(* Logix 5000 project; controller RN21_Architecture 1769-L16ER-BB1B rev 35.11; software revision 35.00 *)
// For Developing the Arch

TASK MainTask (continuous, watchdog 500 ms) : MainProgram

MODULES
   Local : 1769-L16ER-BB1B (PointIO 0, rev 35.11)
      Discrete_IO : Embedded (PointIO 1, rev 35.11, Output RPI 20 ms)
END_MODULES

TYPE UDT_Alarm :
STRUCT
   ALM_YearValue : INT;
   ALM_MonthValue : INT;
   ALM_DayValue : INT;
   ALM_HourValue : INT;
   ALM_MinuteValue : INT;
   ALM_SecondValue : INT;
   ALM_ActionId : INT;
   ALM_Reason : INT;
   ALM_AlarmId1 : DINT;
   ALM_AlarmId2 : DINT;
   ALM_AlarmId3 : DINT;
   ALM_AlarmId4 : DINT;
   ALM_AlarmId5 : DINT;
   ALM_AlarmId6 : DINT;
   ALM_AlarmId7 : DINT;
END_STRUCT
END_TYPE

TYPE UDT_Audit :
STRUCT
   AUD_YearValue : INT;
   AUD_MonthValue : INT;
   AUD_DayValue : INT;
   AUD_HourValue : INT;
   AUD_MinuteValue : INT;
   AUD_SecondValue : INT;
   AUD_ActionId : INT;
   AUD_ReasonId : INT;
   AUD_OldValue : REAL;
   AUD_NewValue : REAL;
   AUD_AppUserId : STRING;
END_STRUCT
END_TYPE

TYPE UDT_Batch :
STRUCT
   BMAN_YearValue : INT;
   BMAN_MonthValue : INT;
   BMAN_DayValue : INT;
   BMAN_HourValue : INT;
   BMAN_MinuteValue : INT;
   BMAN_SecondValue : INT;
   BMAN_BATCH_SIZE : REAL;
   BMAN_BatchStatus : INT;
   BMAN_EXPIR_DATE : INT;
   BMAN_MANFACT_DATE : INT;
   BMAN_EXPIRY_MONTH : INT;
   BMAN_EXPIRY_YEAR : INT;
   BMAN_MANFACT_MONTH : INT;
   BMAN_MANFACT_YEAR : INT;
   BMAN_BATCH_RECIPENAME : STRING;
   BMAN_OPERATOR_CODE : STRING;
   BMAN_PROGRAM_NO : STRING;
   BMAN_TAG_NO : STRING;
   BMAN_LOT_NO : STRING;
   BMAN_PRODUCT_CODE : STRING;
   BMAN_PRODUCT_NAME : STRING;
   BMAN_BATCH_NO : STRING;
END_STRUCT
END_TYPE

TYPE UDT_Login :
STRUCT
   LOGIN_YearValue : INT;
   LOGIN_MonthValue : INT;
   LOGIN_DayValue : INT;
   LOGIN_HourValue : INT;
   LOGIN_MinuteValue : INT;
   LOGIN_SecondValue : INT;
   LOGIN_Reason : INT;
   LOGIN_LoginReason : INT;
   LOGIN_AppUserId : STRING;
END_STRUCT
END_TYPE

TYPE UDT_Process :
STRUCT
   PDL_Year : INT;
   PDL_Month : INT;
   PDL_Date : INT;
   PDL_Hour : INT;
   PDL_Minute : INT;
   PDL_Second : INT;
   PDL_Reason : INT;
   PDL_ActionId : INT;
   PDL_ProcessStatus : INT;
   PDL_CYCLEID : INT;
   PDL_ProcessData : REAL[20];
END_STRUCT
END_TYPE

TYPE UDT_Recipe :
STRUCT
   RP_Year : INT;
   RP_Month : INT;
   RP_Date : INT;
   RP_Hour : INT;
   RP_Minute : INT;
   RP_Second : INT;
   RP_PRINT_INTERVAL : INT;
   RP_CYCLE_ID : INT;
   RP_RecipeData1 : REAL[50];
   RP_RecipeData2 : DINT[50];
END_STRUCT
END_TYPE

ADD_ON_INSTRUCTION AOI_ALM_Arch   (* revision 1.0 *)
VAR_INPUT
   FBI_DataLogTrig : BOOL; {required}   // Trigger Bit for Data Log Generation
END_VAR
VAR_IN_OUT
   FBO_TriggerBit : BOOL; {required}   // Server Trigger Bit
   FBIO_Src : UDT_Alarm; {required}   // Source UDT Data
   FBIO_Ser : UDT_Alarm; {required}   // Server UDT Data
END_VAR
VAR_INPUT
   FBI_PLCServerCommFailed : BOOL; {access None, required}   // PLC to Server Communication Fail Timer Done
END_VAR
VAR_IN_OUT
   FBIO_SerUniqueNum : DINT; {required}   // Server Unique Number(Server UID)
   FBIO_SrcUniqueNum : DINT; {required}   // Source Unique Number (PLC UID)
END_VAR
VAR
   FBL_Prim : UDT_Alarm; {access None}   // Primary UDT Data
   FBL_Buff : UDT_Alarm[100]; {access None}   // Buffer UDT Data
   FBL_Sec : UDT_Alarm; {access None}   // Secondary UDT Data
   FBL_IndexStore : DINT; {access None}   // Index Store Value
   FBL_Bit4 : BOOL; {access None}   // Source to Primary Moved
   FBL_TMR2 : TIMER := (PRE := 1, ACC := 1); {access None}   // Source UID Reset Delay
   FBL_Bit1 : BOOL; {access None}   // Source UID Reseted
   FBL_Bit2 : BOOL; {access None}   // Source UID Less than Server UID
   FBL_Bit6 : BOOL; {access None}   // Data Moving From Secondary to Server
   FBL_TMR3 : TIMER := (PRE := 5000, ACC := 5); {access None}   // Load Movement Delay
   FBL_Bit5 : BOOL; {access None}   // Data Load From Buffer to Secondary Flag
   FBL_IndexLoad : DINT; {access None}   // Index Load Value
   FBL_Bit3 : BOOL; {access None}   // Buffer to Secondary Moved
   FBL_TMR1 : TIMER := (PRE := 5000); {access None}   // Server UID Movement Delay
   FBL_PrimUniqueNum : DINT; {access None}   // Primary Unique Number (PLC UID)
   FBL_BuffUniqueNum : DINT[100]; {access None}   // Buffer Unique Number (PLC UID)
   FBL_SecUniqueNum : DINT; {access None}   // Secondary Unique Number (PLC UID)
   FBL_ONS : DINT; {access None}   // Common ONS DINT
END_VAR

ROUTINE Logic   (* ladder *)
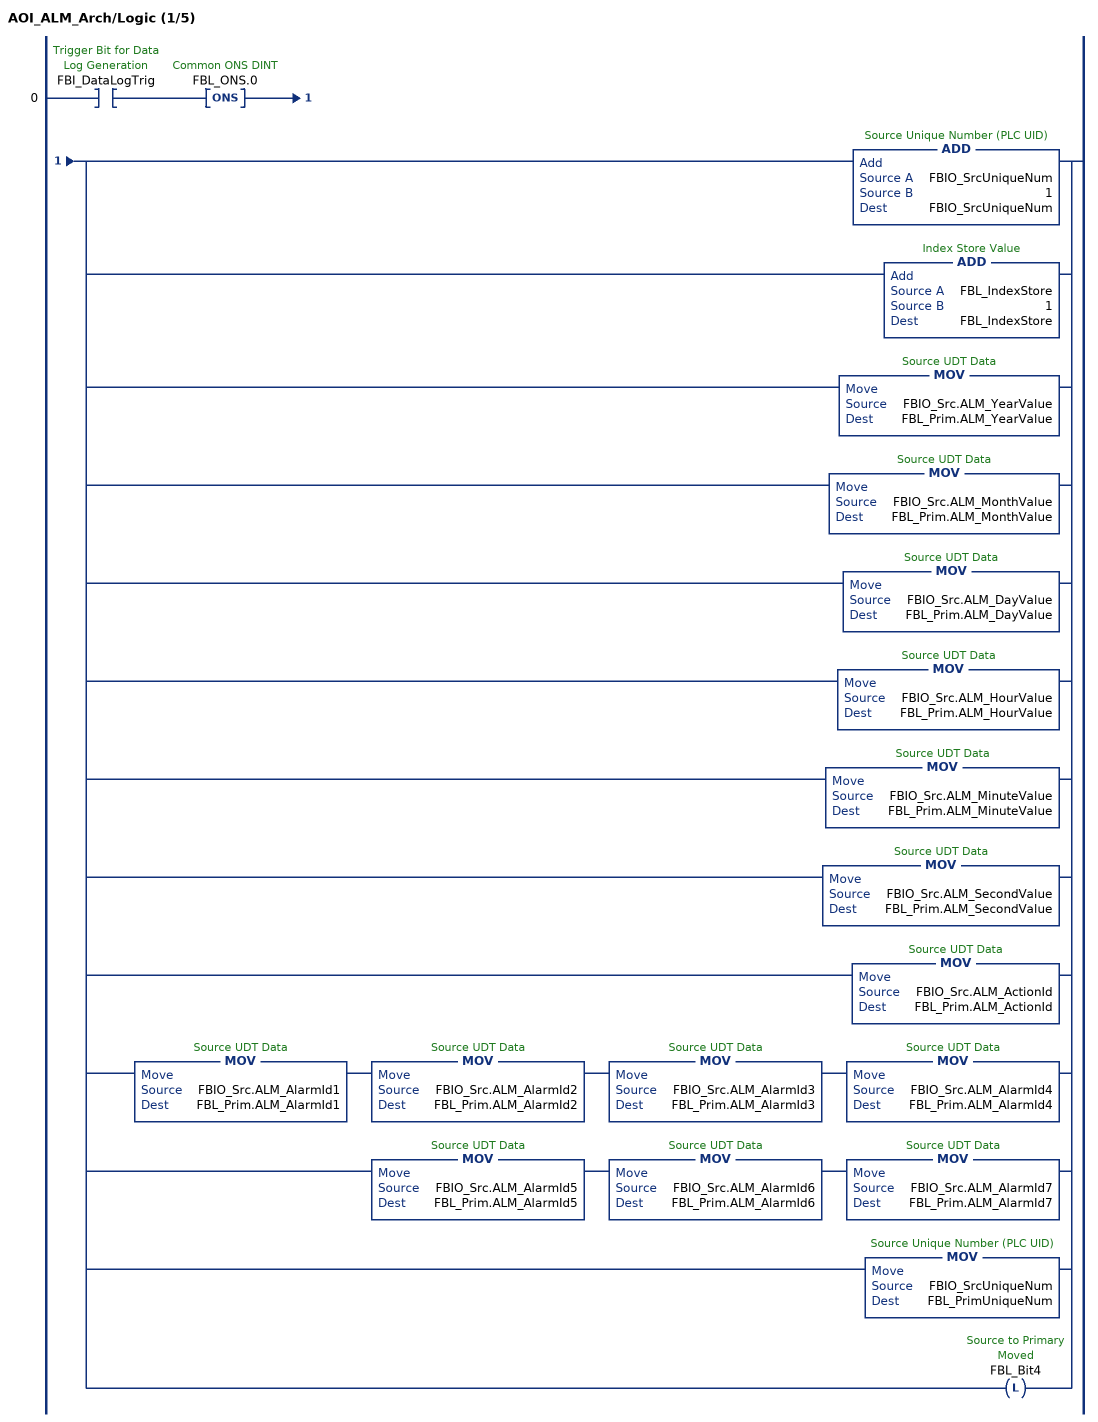
   0: XIC(FBI_DataLogTrig)ONS(FBL_ONS.0)[ADD(FBIO_SrcUniqueNum,1,FBIO_SrcUniqueNum) ,ADD(FBL_IndexStore,1,FBL_IndexStore) ,MOV(FBIO_Src.ALM_YearValue,FBL_Prim.ALM_YearValue) ,MOV(FBIO_Src.ALM_MonthValue,FBL_Prim.ALM_MonthValue) ,MOV(FBIO_Src.ALM_DayValue,FBL_Prim.ALM_DayValue) ,MOV(FBIO_Src.ALM_HourValue,FBL_Prim.ALM_HourValue) ,MOV(FBIO_Src.ALM_MinuteValue,FBL_Prim.ALM_MinuteValue) ,MOV(FBIO_Src.ALM_SecondValue,FBL_Prim.ALM_SecondValue) ,MOV(FBIO_Src.ALM_ActionId,FBL_Prim.ALM_ActionId) ,MOV(FBIO_Src.ALM_AlarmId1,FBL_Prim.ALM_AlarmId1) MOV(FBIO_Src.ALM_AlarmId2,FBL_Prim.ALM_AlarmId2) MOV(FBIO_Src.ALM_AlarmId3,FBL_Prim.ALM_AlarmId3) MOV(FBIO_Src.ALM_AlarmId4,FBL_Prim.ALM_AlarmId4) ,MOV(FBIO_Src.ALM_AlarmId5,FBL_Prim.ALM_AlarmId5) MOV(FBIO_Src.ALM_AlarmId6,FBL_Prim.ALM_AlarmId6) MOV(FBIO_Src.ALM_AlarmId7,FBL_Prim.ALM_AlarmId7) ,MOV(FBIO_SrcUniqueNum,FBL_PrimUniqueNum) ,OTL(FBL_Bit4) ];
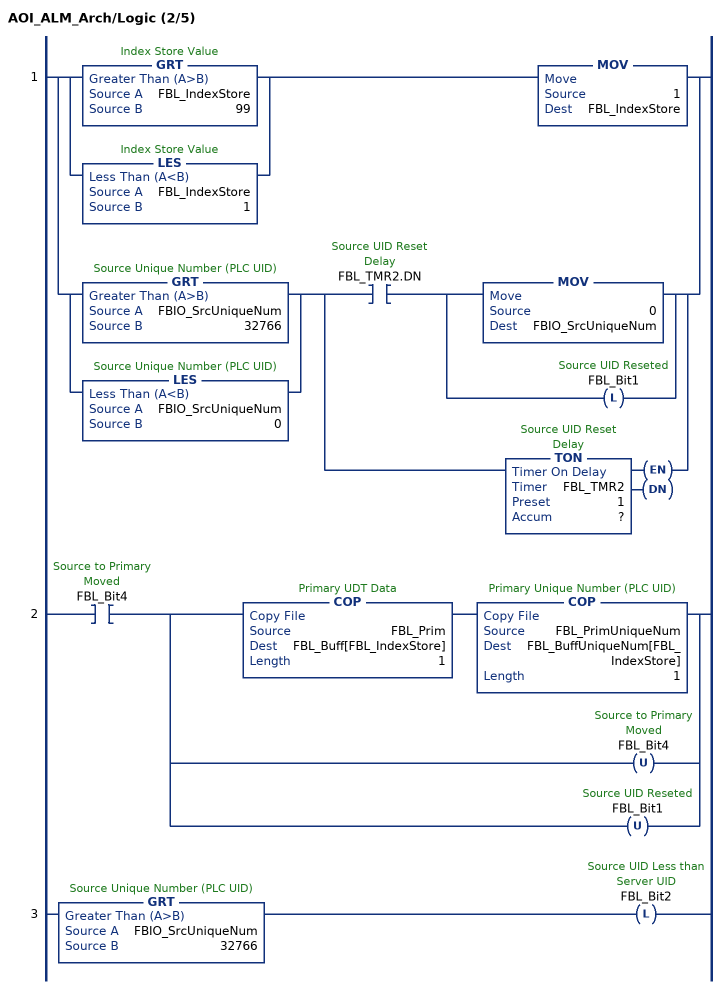
   1: [[GRT(FBL_IndexStore,99) ,LES(FBL_IndexStore,1) ] MOV(1,FBL_IndexStore) ,[GRT(FBIO_SrcUniqueNum,32766) ,LES(FBIO_SrcUniqueNum,0) ] [XIC(FBL_TMR2.DN) [MOV(0,FBIO_SrcUniqueNum) ,OTL(FBL_Bit1) ] ,TON(FBL_TMR2,?,?) ] ];
   2: XIC(FBL_Bit4)[COP(FBL_Prim,FBL_Buff[FBL_IndexStore],1) COP(FBL_PrimUniqueNum,FBL_BuffUniqueNum[FBL_IndexStore],1) ,OTU(FBL_Bit4) ,OTU(FBL_Bit1) ];
   3: GRT(FBIO_SrcUniqueNum,32766)OTL(FBL_Bit2);
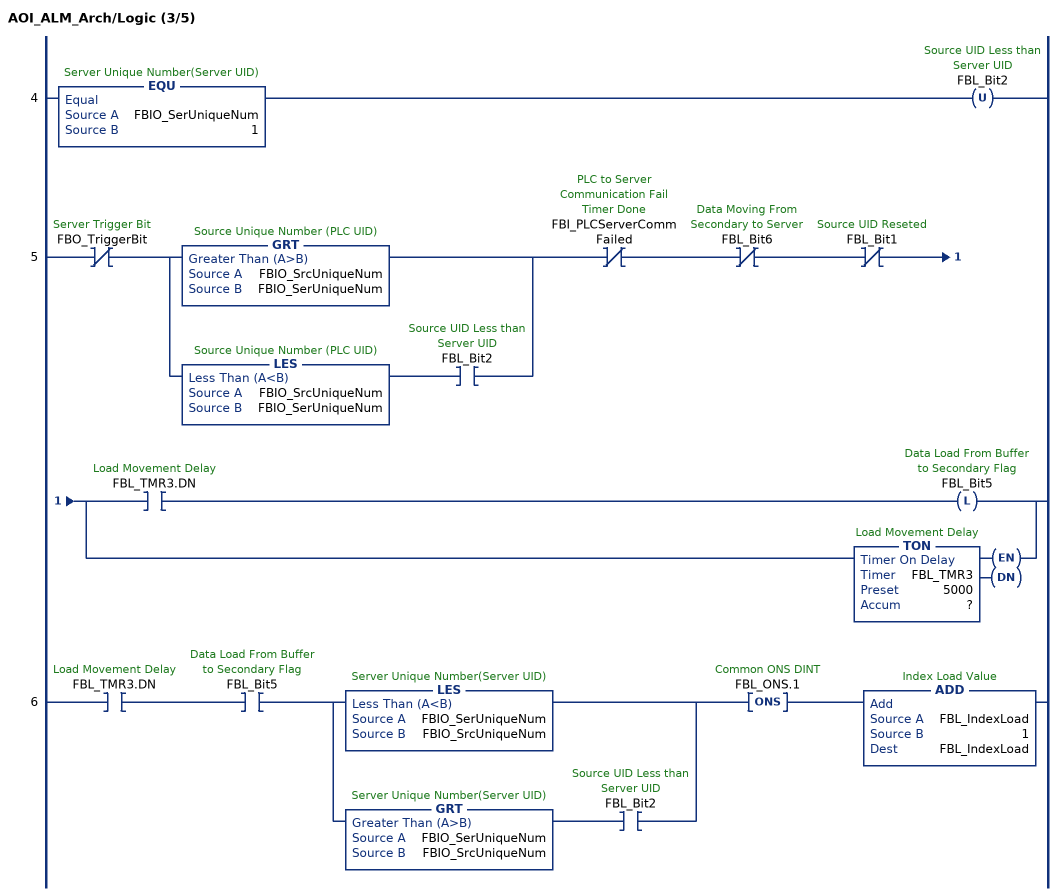
   4: EQU(FBIO_SerUniqueNum,1)OTU(FBL_Bit2);
   5: XIO(FBO_TriggerBit)[GRT(FBIO_SrcUniqueNum,FBIO_SerUniqueNum) ,LES(FBIO_SrcUniqueNum,FBIO_SerUniqueNum) XIC(FBL_Bit2) ]XIO(FBI_PLCServerCommFailed)XIO(FBL_Bit6)XIO(FBL_Bit1)[XIC(FBL_TMR3.DN) OTL(FBL_Bit5) ,TON(FBL_TMR3,?,?) ];
   6: XIC(FBL_TMR3.DN)XIC(FBL_Bit5)[LES(FBIO_SerUniqueNum,FBIO_SrcUniqueNum) ,GRT(FBIO_SerUniqueNum,FBIO_SrcUniqueNum) XIC(FBL_Bit2) ]ONS(FBL_ONS.1)ADD(FBL_IndexLoad,1,FBL_IndexLoad);
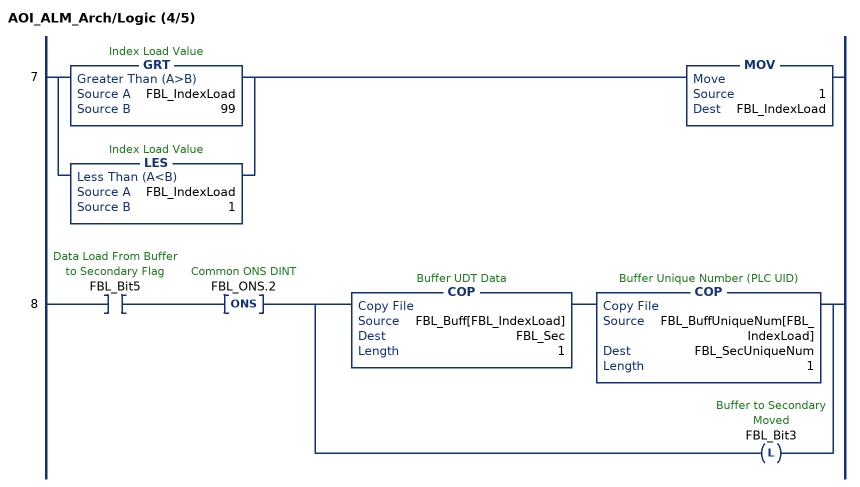
   7: [GRT(FBL_IndexLoad,99) ,LES(FBL_IndexLoad,1) ]MOV(1,FBL_IndexLoad);
   8: XIC(FBL_Bit5)ONS(FBL_ONS.2)[COP(FBL_Buff[FBL_IndexLoad],FBL_Sec,1) COP(FBL_BuffUniqueNum[FBL_IndexLoad],FBL_SecUniqueNum,1) ,OTL(FBL_Bit3) ];
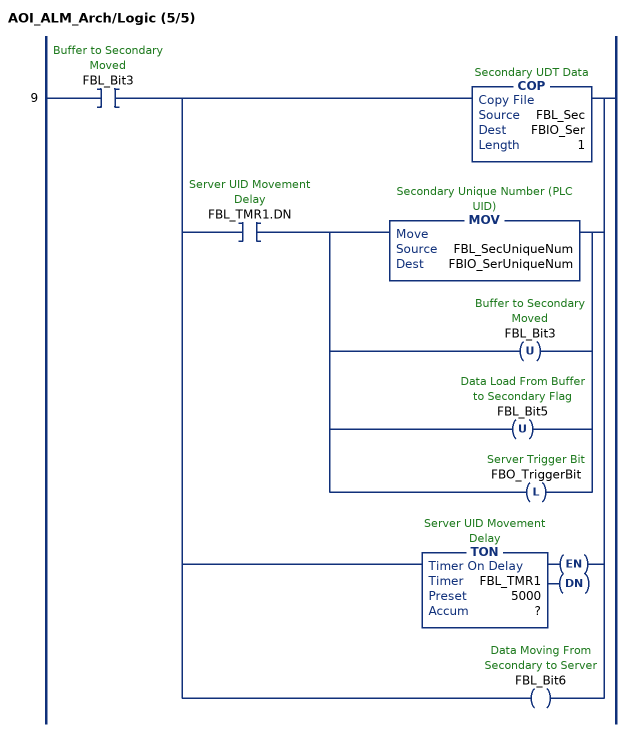
   9: XIC(FBL_Bit3)[COP(FBL_Sec,FBIO_Ser,1) ,XIC(FBL_TMR1.DN) [MOV(FBL_SecUniqueNum,FBIO_SerUniqueNum) ,OTU(FBL_Bit3) ,OTU(FBL_Bit5) ,OTL(FBO_TriggerBit) ] ,TON(FBL_TMR1,?,?) ,OTE(FBL_Bit6) ];
END_ROUTINE
END_ADD_ON_INSTRUCTION

ADD_ON_INSTRUCTION AOI_ALM_DataCapture   (* revision 1.0 *)
// Alarm Data Capture logic
VAR_INPUT
   FBI_AlarmTag : BOOL; {required}
END_VAR
VAR_OUTPUT
   FBO_AlarmPosID : BOOL; {access Read Only, required}
   FBO_ALM_Trig : BOOL; {required}
END_VAR
VAR
   FBL_PosTrig : BOOL; {access None}
   FBL_NegTrig : BOOL; {access None}
   ONS : DINT; {access None}
END_VAR

ROUTINE Logic   (* ladder *)
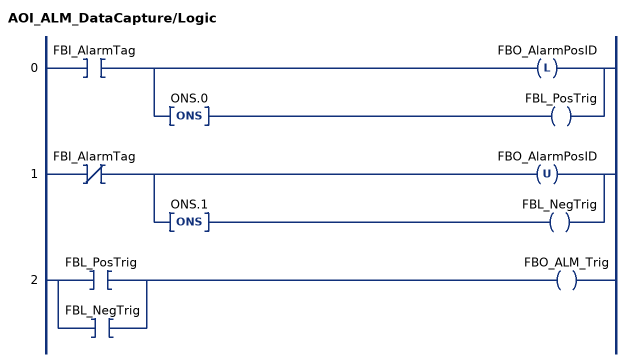
   0: XIC(FBI_AlarmTag)[OTL(FBO_AlarmPosID) ,ONS(ONS.0) OTE(FBL_PosTrig) ];
   1: XIO(FBI_AlarmTag)[OTU(FBO_AlarmPosID) ,ONS(ONS.1) OTE(FBL_NegTrig) ];
   2: [XIC(FBL_PosTrig) ,XIC(FBL_NegTrig) ]OTE(FBO_ALM_Trig);
END_ROUTINE
END_ADD_ON_INSTRUCTION

ADD_ON_INSTRUCTION AOI_AUD_Arch   (* revision 1.0 *)
VAR_INPUT
   FBI_DataLogTrig : BOOL; {required}   // Trigger Bit for Data Log Generation
END_VAR
VAR_IN_OUT
   FBO_TriggerBit : BOOL; {required}   // Server Trigger Bit
   FBIO_Src : UDT_Audit; {required}   // Source UDT Data
   FBIO_Ser : UDT_Audit; {required}   // Server UDT Data
END_VAR
VAR_INPUT
   FBI_PLCServerCommFailed : BOOL; {access None, required}   // PLC to Server Communication Fail Timer Done
END_VAR
VAR_IN_OUT
   FBIO_SrcUniqueNum : DINT; {required}   // Source Unique Number(PLC UID)
   FBIO_SerUniqueNum : DINT; {required}   // Server Unique Number(PLC UID)
END_VAR
VAR
   FBL_Prim : UDT_Audit; {access None}   // Primary UDT Data
   FBL_Buff : UDT_Audit[100]; {access None}   // Buffer UDT Data
   FBL_Sec : UDT_Audit; {access None}   // Secondary UDT Data
   FBL_IndexStore : DINT; {access None}   // Index Store Value
   FBL_Bit4 : BOOL; {access None}   // Primary Movement Completed
   FBL_TMR2 : TIMER := (PRE := 1, ACC := 1); {access None}   // Source UID Reset Delay
   FBL_Bit1 : BOOL; {access None}   // Source UID Reset
   FBL_Bit2 : BOOL; {access None}   // Source UID Less than Server UID
   FBL_Bit6 : BOOL; {access None}   // Data Moving From Secondary to Server
   FBL_TMR3 : TIMER := (PRE := 5000, ACC := 5); {access None}   // Load Movement Delay
   FBL_Bit5 : BOOL; {access None}   // Data Load From Buffer to Secondary Flag
   FBL_IndexLoad : DINT; {access None}   // Index Load Value
   FBL_Bit3 : BOOL; {access None}   // Secondary Movement Completed
   FBL_TMR1 : TIMER := (PRE := 5000); {access None}   // Server UID Movement Delay
   FBL_PrimUniqueNum : DINT; {access None}   // Primary Unique Number (PLC UID)
   FBL_SecUniqueNum : DINT; {access None}   // Secondary Unique Number(PLC UID)
   FBL_BuffUniqueNum : DINT[100]; {access None}   // Buffer Unique Number(PLC UID)
   FBL_ONS : DINT; {access None}   // Common ONS DINT
END_VAR

ROUTINE Logic   (* ladder *)
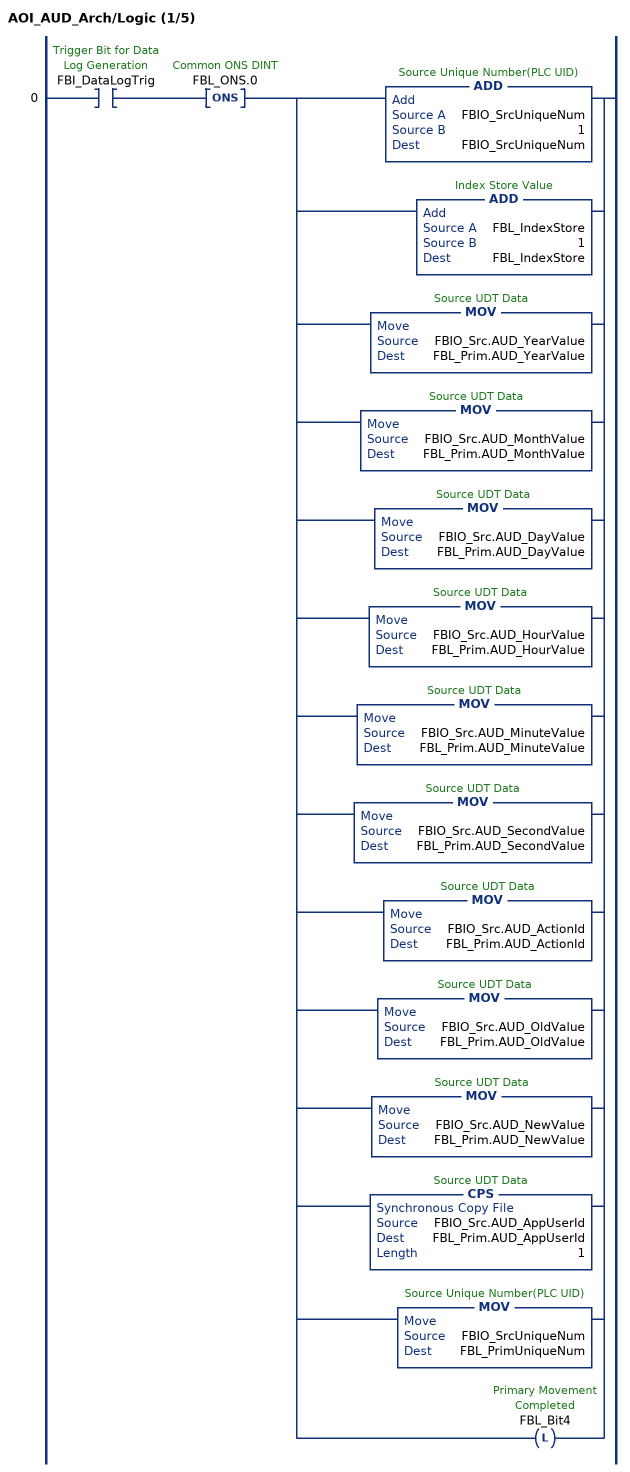
   0: XIC(FBI_DataLogTrig)ONS(FBL_ONS.0)[ADD(FBIO_SrcUniqueNum,1,FBIO_SrcUniqueNum) ,ADD(FBL_IndexStore,1,FBL_IndexStore) ,MOV(FBIO_Src.AUD_YearValue,FBL_Prim.AUD_YearValue) ,MOV(FBIO_Src.AUD_MonthValue,FBL_Prim.AUD_MonthValue) ,MOV(FBIO_Src.AUD_DayValue,FBL_Prim.AUD_DayValue) ,MOV(FBIO_Src.AUD_HourValue,FBL_Prim.AUD_HourValue) ,MOV(FBIO_Src.AUD_MinuteValue,FBL_Prim.AUD_MinuteValue) ,MOV(FBIO_Src.AUD_SecondValue,FBL_Prim.AUD_SecondValue) ,MOV(FBIO_Src.AUD_ActionId,FBL_Prim.AUD_ActionId) ,MOV(FBIO_Src.AUD_OldValue,FBL_Prim.AUD_OldValue) ,MOV(FBIO_Src.AUD_NewValue,FBL_Prim.AUD_NewValue) ,CPS(FBIO_Src.AUD_AppUserId,FBL_Prim.AUD_AppUserId,1) ,MOV(FBIO_SrcUniqueNum,FBL_PrimUniqueNum) ,OTL(FBL_Bit4) ];
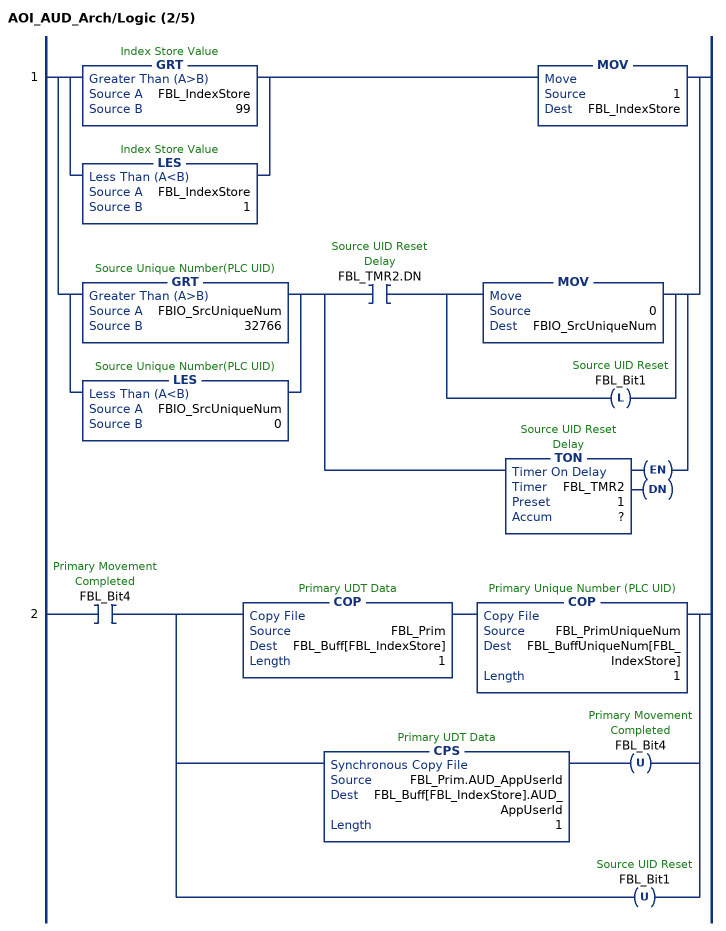
   1: [[GRT(FBL_IndexStore,99) ,LES(FBL_IndexStore,1) ] MOV(1,FBL_IndexStore) ,[GRT(FBIO_SrcUniqueNum,32766) ,LES(FBIO_SrcUniqueNum,0) ] [XIC(FBL_TMR2.DN) [MOV(0,FBIO_SrcUniqueNum) ,OTL(FBL_Bit1) ] ,TON(FBL_TMR2,?,?) ] ];
   2: XIC(FBL_Bit4)[COP(FBL_Prim,FBL_Buff[FBL_IndexStore],1) COP(FBL_PrimUniqueNum,FBL_BuffUniqueNum[FBL_IndexStore],1) ,CPS(FBL_Prim.AUD_AppUserId,FBL_Buff[FBL_IndexStore].AUD_AppUserId,1) OTU(FBL_Bit4) ,OTU(FBL_Bit1) ];
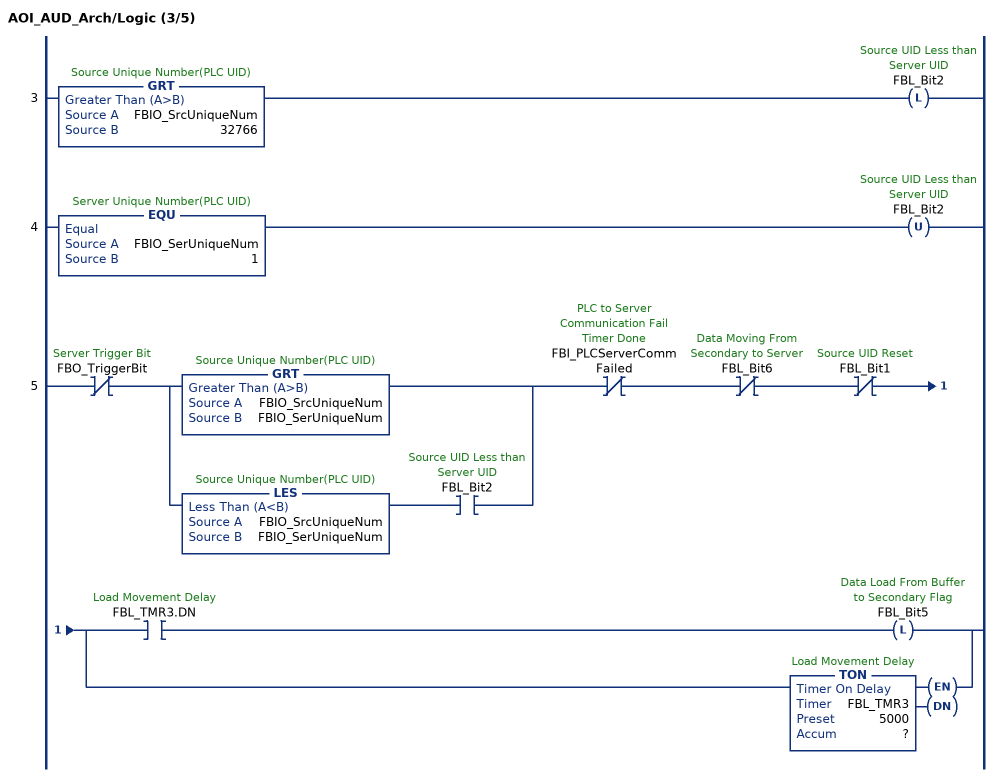
   3: GRT(FBIO_SrcUniqueNum,32766)OTL(FBL_Bit2);
   4: EQU(FBIO_SerUniqueNum,1)OTU(FBL_Bit2);
   5: XIO(FBO_TriggerBit)[GRT(FBIO_SrcUniqueNum,FBIO_SerUniqueNum) ,LES(FBIO_SrcUniqueNum,FBIO_SerUniqueNum) XIC(FBL_Bit2) ]XIO(FBI_PLCServerCommFailed)XIO(FBL_Bit6)XIO(FBL_Bit1)[XIC(FBL_TMR3.DN) OTL(FBL_Bit5) ,TON(FBL_TMR3,?,?) ];
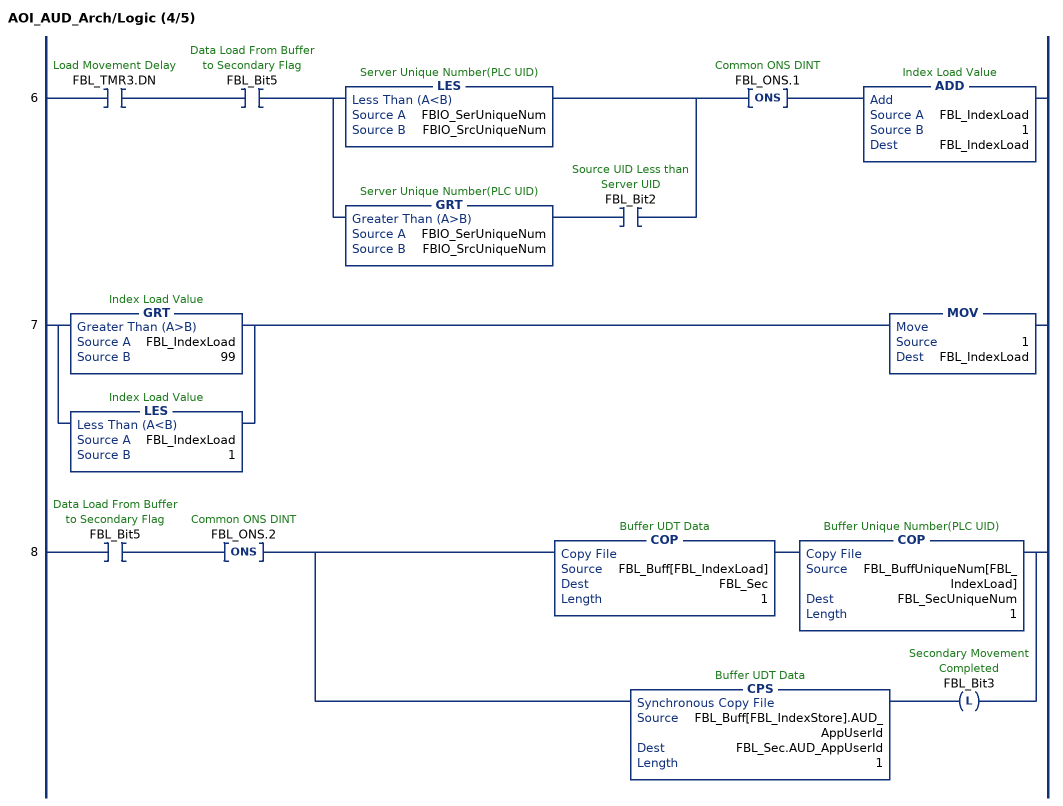
   6: XIC(FBL_TMR3.DN)XIC(FBL_Bit5)[LES(FBIO_SerUniqueNum,FBIO_SrcUniqueNum) ,GRT(FBIO_SerUniqueNum,FBIO_SrcUniqueNum) XIC(FBL_Bit2) ]ONS(FBL_ONS.1)ADD(FBL_IndexLoad,1,FBL_IndexLoad);
   7: [GRT(FBL_IndexLoad,99) ,LES(FBL_IndexLoad,1) ]MOV(1,FBL_IndexLoad);
   8: XIC(FBL_Bit5)ONS(FBL_ONS.2)[COP(FBL_Buff[FBL_IndexLoad],FBL_Sec,1) COP(FBL_BuffUniqueNum[FBL_IndexLoad],FBL_SecUniqueNum,1) ,CPS(FBL_Buff[FBL_IndexStore].AUD_AppUserId,FBL_Sec.AUD_AppUserId,1) OTL(FBL_Bit3) ];
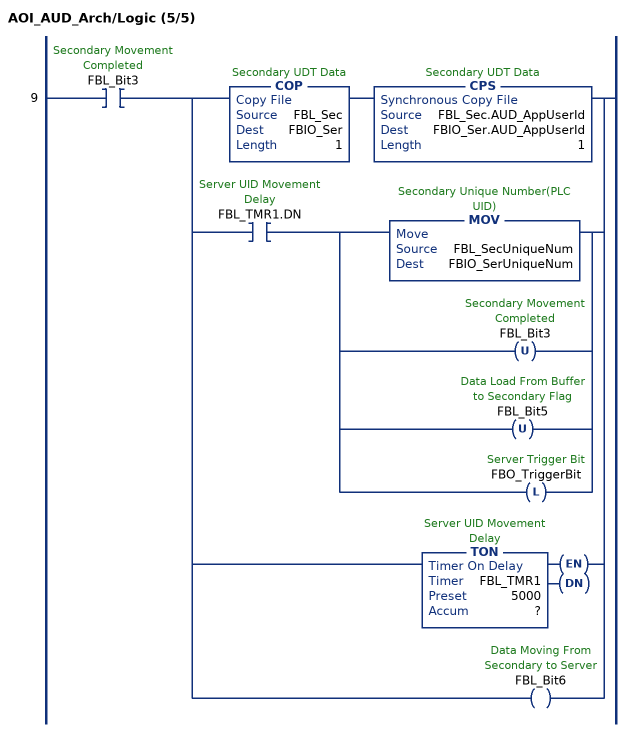
   9: XIC(FBL_Bit3)[COP(FBL_Sec,FBIO_Ser,1) CPS(FBL_Sec.AUD_AppUserId,FBIO_Ser.AUD_AppUserId,1) ,XIC(FBL_TMR1.DN) [MOV(FBL_SecUniqueNum,FBIO_SerUniqueNum) ,OTU(FBL_Bit3) ,OTU(FBL_Bit5) ,OTL(FBO_TriggerBit) ] ,TON(FBL_TMR1,?,?) ,OTE(FBL_Bit6) ];
END_ROUTINE
END_ADD_ON_INSTRUCTION

ADD_ON_INSTRUCTION AOI_AUD_DataCapture1   (* revision 1.0 *)
// AuditData Capture logic for Momentary Button Action
VAR_INPUT
   FBI_BAM : BOOL; {required}
END_VAR
VAR_OUTPUT
   FBO_AUD_Trig : BOOL; {access Read Only, required}
   FBO_ActionID : INT; {access Read Only, required}
END_VAR
VAR_INPUT
   FBI_ActionID : INT; {required}
END_VAR
VAR_OUTPUT
   FBO_OldValue : REAL; {access Read Only, required}
   FBO_NewValue : REAL; {access Read Only, required}
END_VAR
VAR
   FBL_ONS : DINT; {access None}
END_VAR

ROUTINE Logic   (* ladder *)
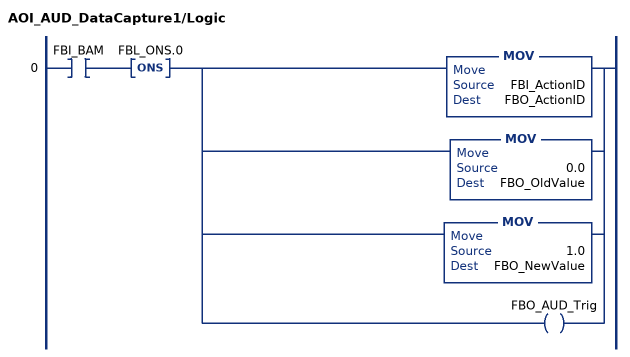
   0: XIC(FBI_BAM)ONS(FBL_ONS.0)[MOV(FBI_ActionID,FBO_ActionID) ,MOV(0.0,FBO_OldValue) ,MOV(1.0,FBO_NewValue) ,OTE(FBO_AUD_Trig) ];
END_ROUTINE
END_ADD_ON_INSTRUCTION

ADD_ON_INSTRUCTION AOI_AUD_DataCapture2   (* revision 1.0 *)
// Audit Data Capture logic for Toggle Button Action
VAR_INPUT
   FBI_BAT : BOOL; {required}
END_VAR
VAR_OUTPUT
   FBO_AUD_Trig : BOOL; {access Read Only, required}
   FBO_ActionID : INT; {access Read Only, required}
END_VAR
VAR_INPUT
   FBI_ActionID : INT; {required}
END_VAR
VAR_OUTPUT
   FBO_OldValue : REAL; {access Read Only, required}
   FBO_NewValue : REAL; {access Read Only, required}
END_VAR
VAR
   FBL_PosTrig : BOOL; {access None}
   FBL_NegTrig : BOOL; {access None}
   FBL_ONS : DINT; {access None}
END_VAR

ROUTINE Logic   (* ladder *)
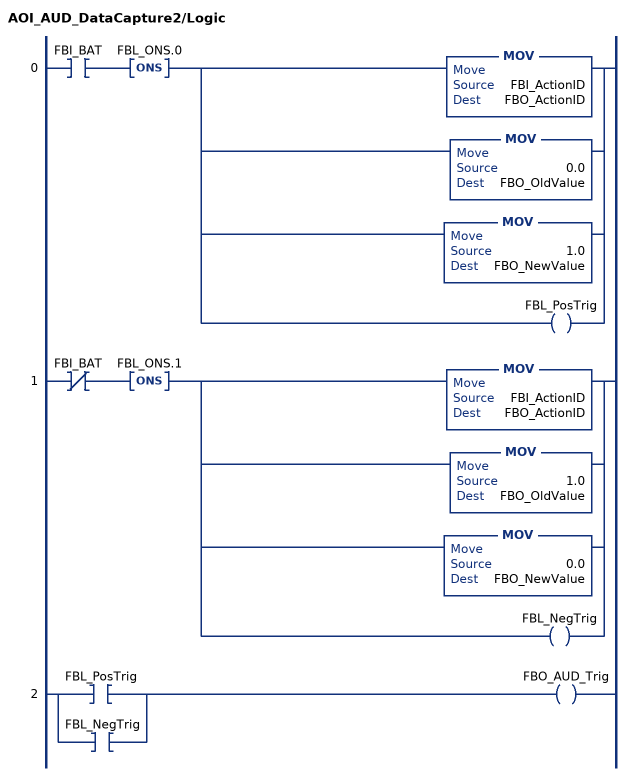
   0: XIC(FBI_BAT)ONS(FBL_ONS.0)[MOV(FBI_ActionID,FBO_ActionID) ,MOV(0.0,FBO_OldValue) ,MOV(1.0,FBO_NewValue) ,OTE(FBL_PosTrig) ];
   1: XIO(FBI_BAT)ONS(FBL_ONS.1)[MOV(FBI_ActionID,FBO_ActionID) ,MOV(1.0,FBO_OldValue) ,MOV(0.0,FBO_NewValue) ,OTE(FBL_NegTrig) ];
   2: [XIC(FBL_PosTrig) ,XIC(FBL_NegTrig) ]OTE(FBO_AUD_Trig);
END_ROUTINE
END_ADD_ON_INSTRUCTION

ADD_ON_INSTRUCTION AOI_AUD_DataCapture3   (* revision 1.0 *)
// Audit Data Capture logic for Numeric Entry
VAR_INPUT
   FBI_NE : REAL; {required}
   FBI_ActionID : INT; {required}
END_VAR
VAR_OUTPUT
   FBO_AUD_TRIG : BOOL; {required}
   FBO_OldValue : REAL; {access Read Only, required}
   FBO_NewValue : REAL; {access Read Only, required}
   FBO_ActionID : INT; {access Read Only, required}
END_VAR
VAR
   FBL_NEWVALUE : REAL; {access None}
   FBL_OLDVALUE : REAL; {access None}
   TMR_DataMovDly : TIMER := (PRE := 20); {access None}   // Delay Timer to Move the Values
   FBL_ONS : DINT; {access None}
END_VAR

ROUTINE Logic   (* ladder *)
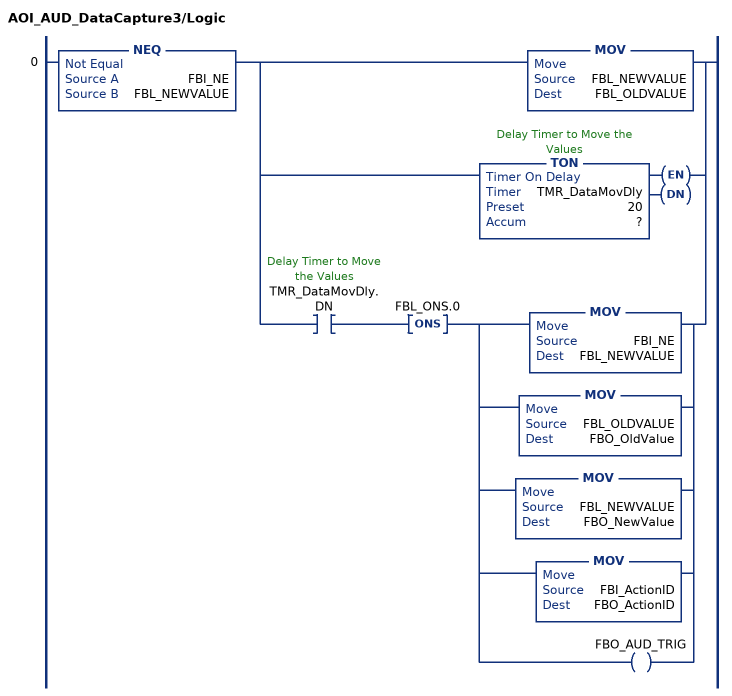
   0: NEQ(FBI_NE,FBL_NEWVALUE)[MOV(FBL_NEWVALUE,FBL_OLDVALUE) ,TON(TMR_DataMovDly,?,?) ,XIC(TMR_DataMovDly.DN) ONS(FBL_ONS.0) [MOV(FBI_NE,FBL_NEWVALUE) ,MOV(FBL_OLDVALUE,FBO_OldValue) ,MOV(FBL_NEWVALUE,FBO_NewValue) ,MOV(FBI_ActionID,FBO_ActionID) ,OTE(FBO_AUD_TRIG) ] ];
END_ROUTINE
END_ADD_ON_INSTRUCTION

ADD_ON_INSTRUCTION AOI_BMAN_Arch   (* revision 1.0 *)
VAR_INPUT
   FBI_DataLogTrig : BOOL; {required}   // Trigger Bit for Data Log Generation
END_VAR
VAR_IN_OUT
   FBO_TriggerBit : BOOL; {required}   // Server Trigger Bit
   FBIO_Src : UDT_Batch; {required}   // Source UDT Data
   FBIO_Ser : UDT_Batch; {required}   // Server UDT Data
END_VAR
VAR_INPUT
   FBI_PLCServerCommFailed : BOOL; {access None, required}   // PLC to Server Communication Fail Timer Done
END_VAR
VAR_IN_OUT
   FBIO_SrcUniqueNum : DINT; {required}   // Source Unique Number (PLC UID)
   FBIO_SerUniqueNum : DINT; {required}   // Server Unique Number (PLC UID)
END_VAR
VAR
   FBL_Prim : UDT_Batch; {access None}   // Primary UDT Data
   FBL_Buff : UDT_Batch[5]; {access None}   // Buffer UDT Data
   FBL_Sec : UDT_Batch; {access None}   // Secondary UDT Data
   FBL_IndexStore : DINT; {access None}   // Index Store
   FBL_Bit4 : BOOL; {access None}   // Primary Movement Completed
   FBL_TMR2 : TIMER := (PRE := 1, ACC := 1); {access None}   // Source UID Reset Delay
   FBL_Bit1 : BOOL; {access None}   // Source UID Reset
   FBL_Bit2 : BOOL; {access None}   // Source UID Less than Server UID
   FBL_Bit6 : BOOL; {access None}   // Data Moving From Secondary to Server
   FBL_TMR3 : TIMER := (PRE := 5000, ACC := 5); {access None}   // Load Movement Delay
   FBL_Bit5 : BOOL; {access None}   // Data Load From Buffer to Secondary Flag
   FBL_IndexLoad : DINT; {access None}   // Index Load
   FBL_Bit3 : BOOL; {access None}   // Secondary Movement Completed
   FBL_TMR1 : TIMER := (PRE := 5000); {access None}   // Server UID Movement Delay
   FBL_BuffUniqueNum : DINT[5]; {access None}   // Buffer Unique Number (PLC UID)
   FBL_PrimUniqueNum : DINT; {access None}   // Primary Unique Number (PLC UID)
   FBL_SecUniqueNum : DINT; {access None}   // Secondary Unique Number (PLC UID)
   FBL_ONS : DINT; {access None}   // Common ONS DINT
END_VAR

ROUTINE Logic   (* ladder *)
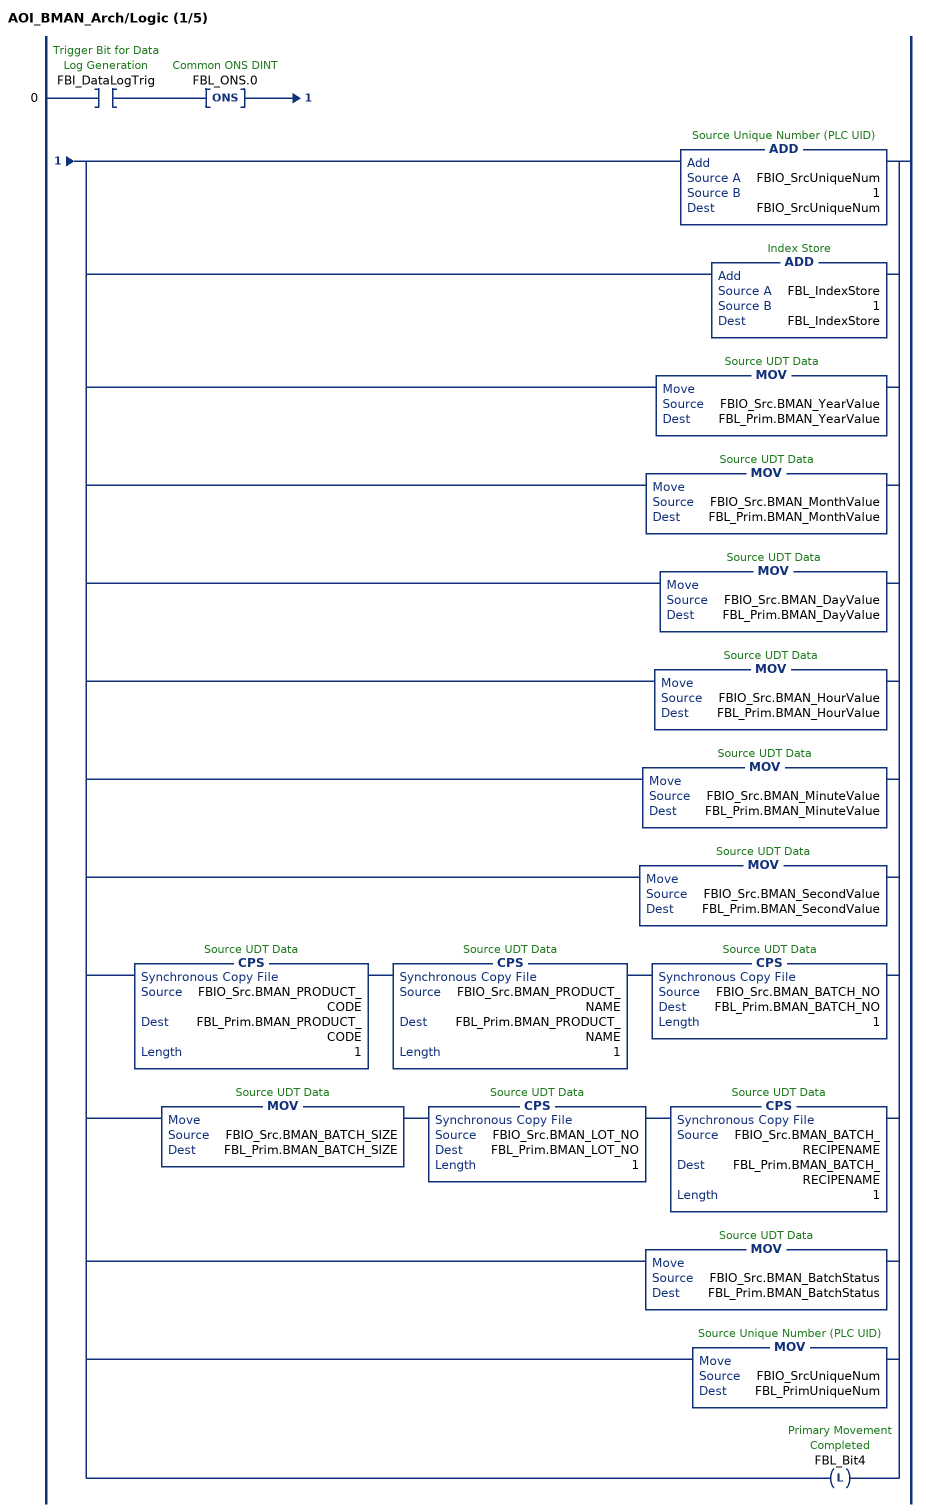
   0: XIC(FBI_DataLogTrig)ONS(FBL_ONS.0)[ADD(FBIO_SrcUniqueNum,1,FBIO_SrcUniqueNum) ,ADD(FBL_IndexStore,1,FBL_IndexStore) ,MOV(FBIO_Src.BMAN_YearValue,FBL_Prim.BMAN_YearValue) ,MOV(FBIO_Src.BMAN_MonthValue,FBL_Prim.BMAN_MonthValue) ,MOV(FBIO_Src.BMAN_DayValue,FBL_Prim.BMAN_DayValue) ,MOV(FBIO_Src.BMAN_HourValue,FBL_Prim.BMAN_HourValue) ,MOV(FBIO_Src.BMAN_MinuteValue,FBL_Prim.BMAN_MinuteValue) ,MOV(FBIO_Src.BMAN_SecondValue,FBL_Prim.BMAN_SecondValue) ,CPS(FBIO_Src.BMAN_PRODUCT_CODE,FBL_Prim.BMAN_PRODUCT_CODE,1) CPS(FBIO_Src.BMAN_PRODUCT_NAME,FBL_Prim.BMAN_PRODUCT_NAME,1) CPS(FBIO_Src.BMAN_BATCH_NO,FBL_Prim.BMAN_BATCH_NO,1) ,MOV(FBIO_Src.BMAN_BATCH_SIZE,FBL_Prim.BMAN_BATCH_SIZE) CPS(FBIO_Src.BMAN_LOT_NO,FBL_Prim.BMAN_LOT_NO,1) CPS(FBIO_Src.BMAN_BATCH_RECIPENAME,FBL_Prim.BMAN_BATCH_RECIPENAME,1) ,MOV(FBIO_Src.BMAN_BatchStatus,FBL_Prim.BMAN_BatchStatus) ,MOV(FBIO_SrcUniqueNum,FBL_PrimUniqueNum) ,OTL(FBL_Bit4) ];
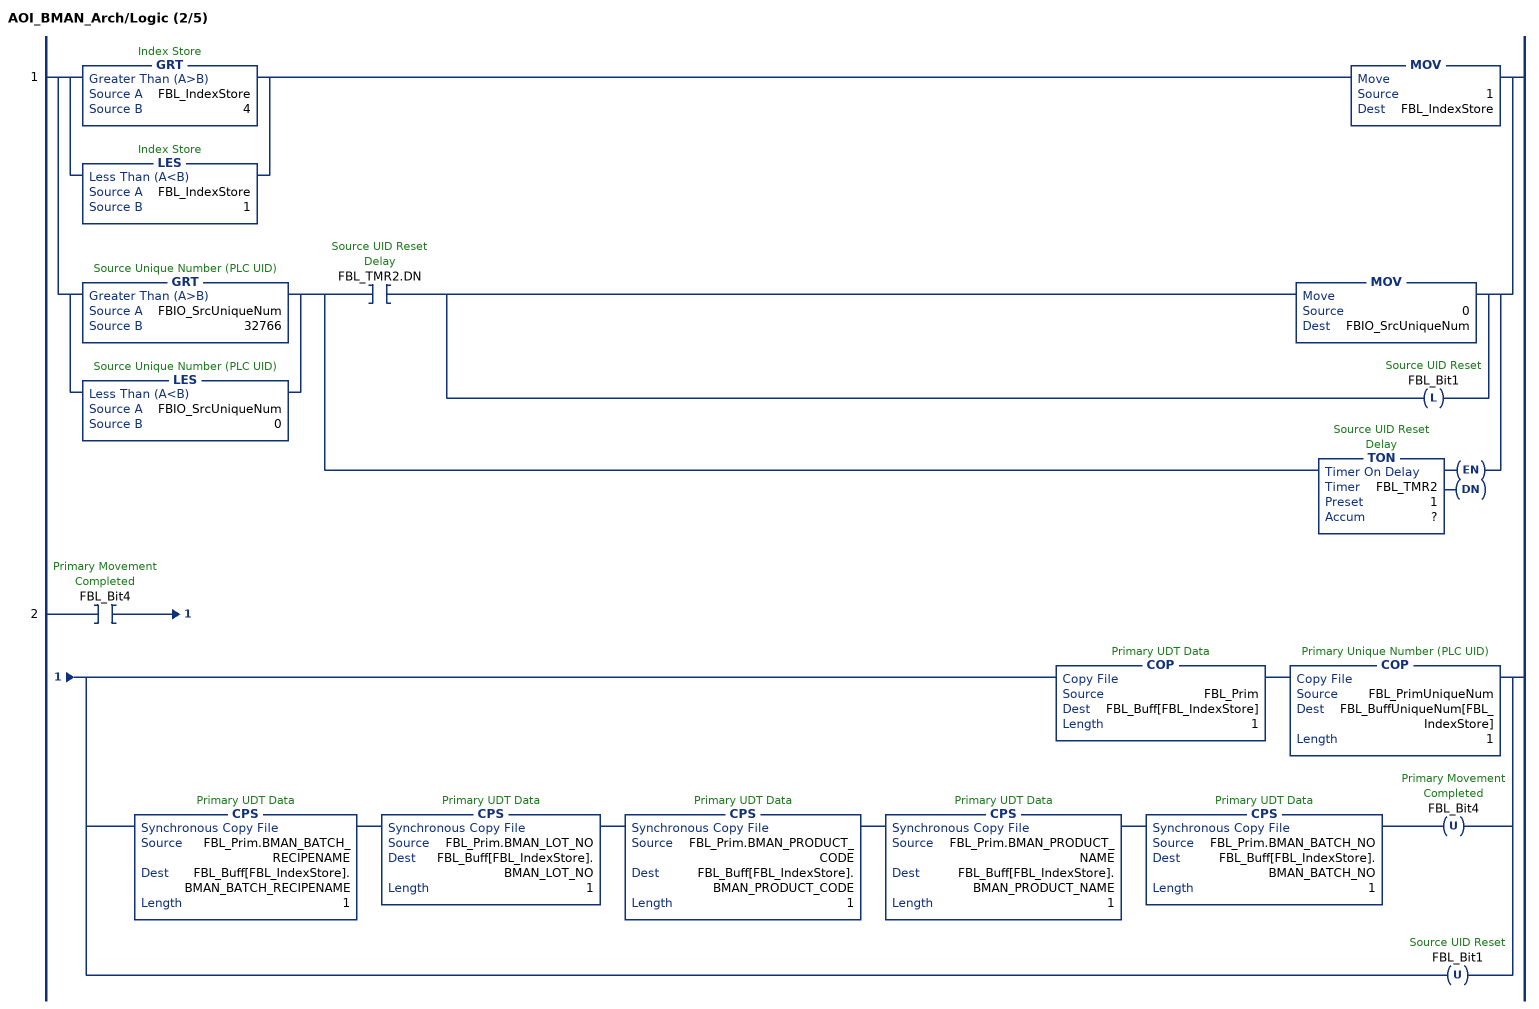
   1: [[GRT(FBL_IndexStore,4) ,LES(FBL_IndexStore,1) ] MOV(1,FBL_IndexStore) ,[GRT(FBIO_SrcUniqueNum,32766) ,LES(FBIO_SrcUniqueNum,0) ] [XIC(FBL_TMR2.DN) [MOV(0,FBIO_SrcUniqueNum) ,OTL(FBL_Bit1) ] ,TON(FBL_TMR2,?,?) ] ];
   2: XIC(FBL_Bit4)[COP(FBL_Prim,FBL_Buff[FBL_IndexStore],1) COP(FBL_PrimUniqueNum,FBL_BuffUniqueNum[FBL_IndexStore],1) ,CPS(FBL_Prim.BMAN_BATCH_RECIPENAME,FBL_Buff[FBL_IndexStore].BMAN_BATCH_RECIPENAME,1) CPS(FBL_Prim.BMAN_LOT_NO,FBL_Buff[FBL_IndexStore].BMAN_LOT_NO,1) CPS(FBL_Prim.BMAN_PRODUCT_CODE,FBL_Buff[FBL_IndexStore].BMAN_PRODUCT_CODE,1) CPS(FBL_Prim.BMAN_PRODUCT_NAME,FBL_Buff[FBL_IndexStore].BMAN_PRODUCT_NAME,1) CPS(FBL_Prim.BMAN_BATCH_NO,FBL_Buff[FBL_IndexStore].BMAN_BATCH_NO,1) OTU(FBL_Bit4) ,OTU(FBL_Bit1) ];
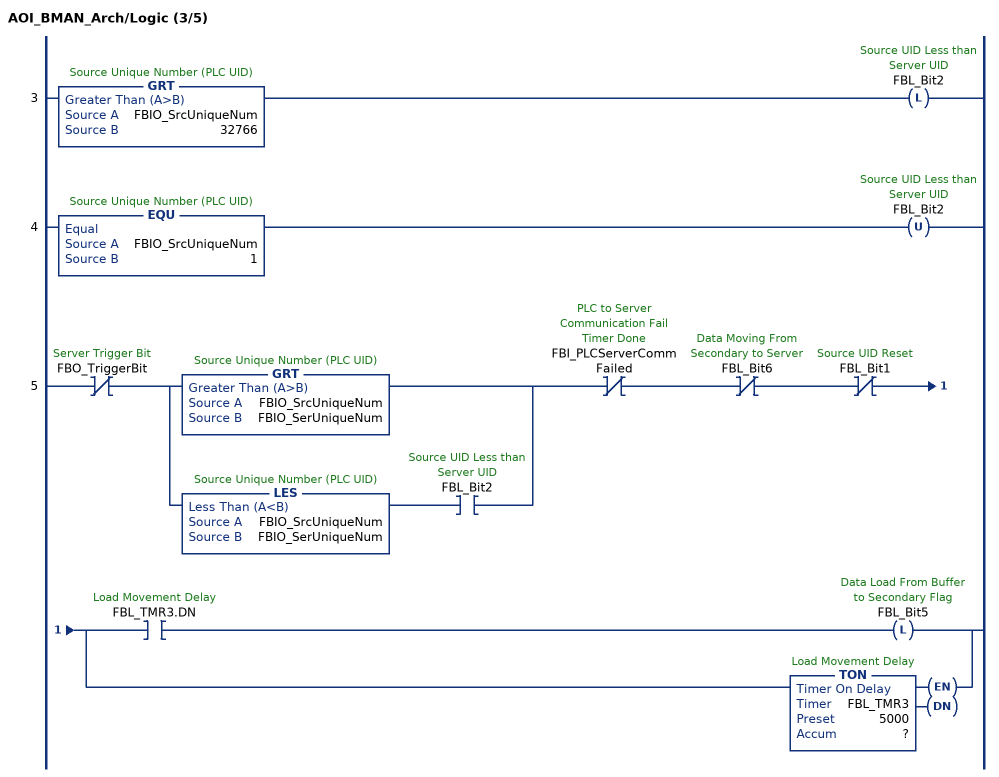
   3: GRT(FBIO_SrcUniqueNum,32766)OTL(FBL_Bit2);
   4: EQU(FBIO_SrcUniqueNum,1)OTU(FBL_Bit2);
   5: XIO(FBO_TriggerBit)[GRT(FBIO_SrcUniqueNum,FBIO_SerUniqueNum) ,LES(FBIO_SrcUniqueNum,FBIO_SerUniqueNum) XIC(FBL_Bit2) ]XIO(FBI_PLCServerCommFailed)XIO(FBL_Bit6)XIO(FBL_Bit1)[XIC(FBL_TMR3.DN) OTL(FBL_Bit5) ,TON(FBL_TMR3,?,?) ];
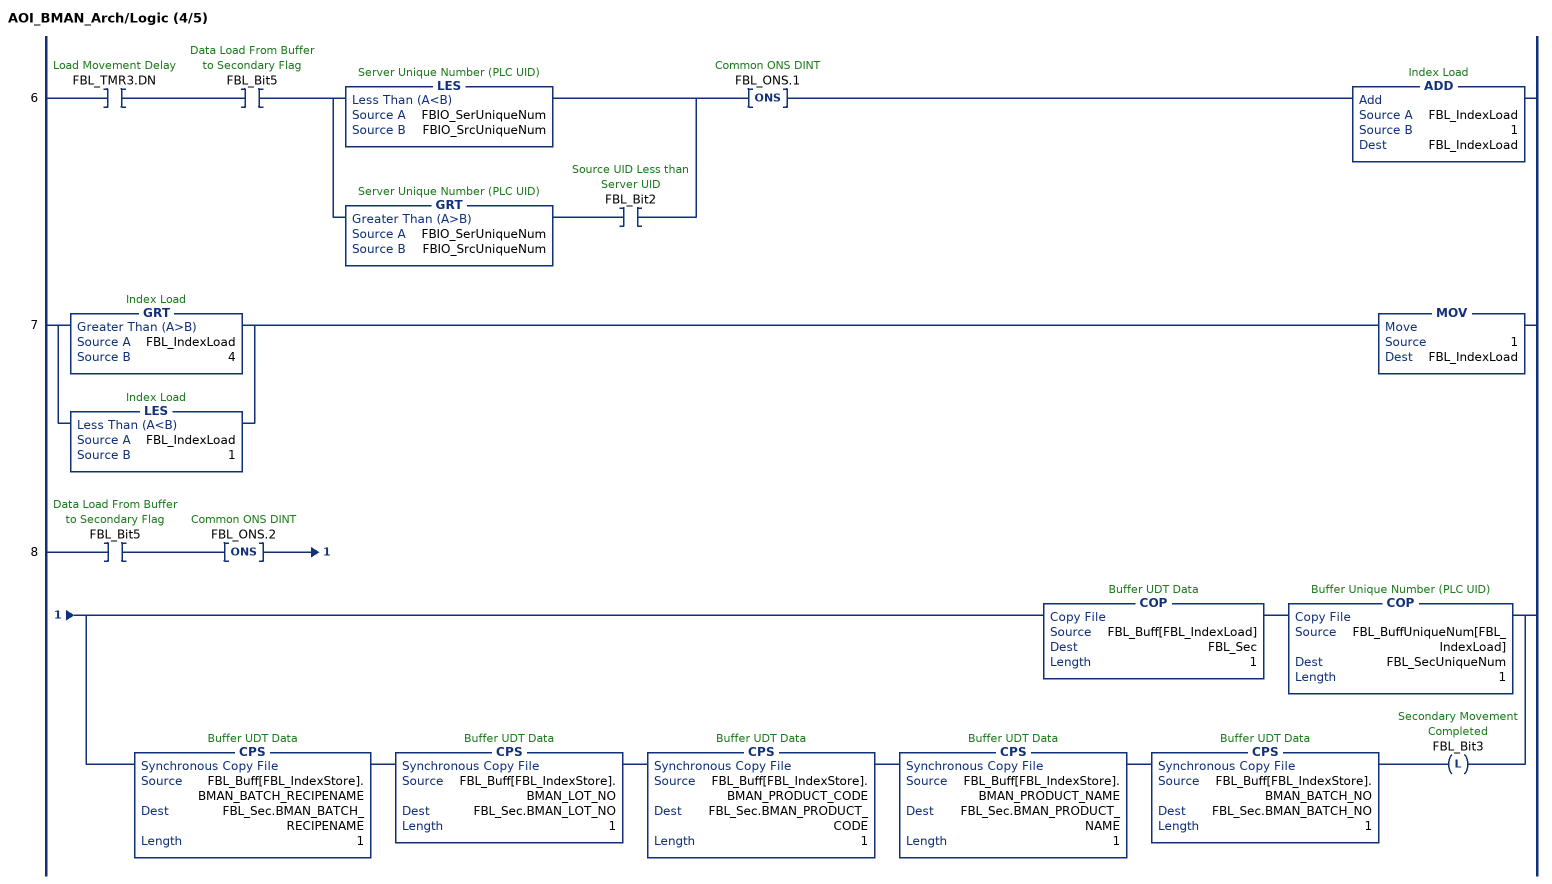
   6: XIC(FBL_TMR3.DN)XIC(FBL_Bit5)[LES(FBIO_SerUniqueNum,FBIO_SrcUniqueNum) ,GRT(FBIO_SerUniqueNum,FBIO_SrcUniqueNum) XIC(FBL_Bit2) ]ONS(FBL_ONS.1)ADD(FBL_IndexLoad,1,FBL_IndexLoad);
   7: [GRT(FBL_IndexLoad,4) ,LES(FBL_IndexLoad,1) ]MOV(1,FBL_IndexLoad);
   8: XIC(FBL_Bit5)ONS(FBL_ONS.2)[COP(FBL_Buff[FBL_IndexLoad],FBL_Sec,1) COP(FBL_BuffUniqueNum[FBL_IndexLoad],FBL_SecUniqueNum,1) ,CPS(FBL_Buff[FBL_IndexStore].BMAN_BATCH_RECIPENAME,FBL_Sec.BMAN_BATCH_RECIPENAME,1) CPS(FBL_Buff[FBL_IndexStore].BMAN_LOT_NO,FBL_Sec.BMAN_LOT_NO,1) CPS(FBL_Buff[FBL_IndexStore].BMAN_PRODUCT_CODE,FBL_Sec.BMAN_PRODUCT_CODE,1) CPS(FBL_Buff[FBL_IndexStore].BMAN_PRODUCT_NAME,FBL_Sec.BMAN_PRODUCT_NAME,1) CPS(FBL_Buff[FBL_IndexStore].BMAN_BATCH_NO,FBL_Sec.BMAN_BATCH_NO,1) OTL(FBL_Bit3) ];
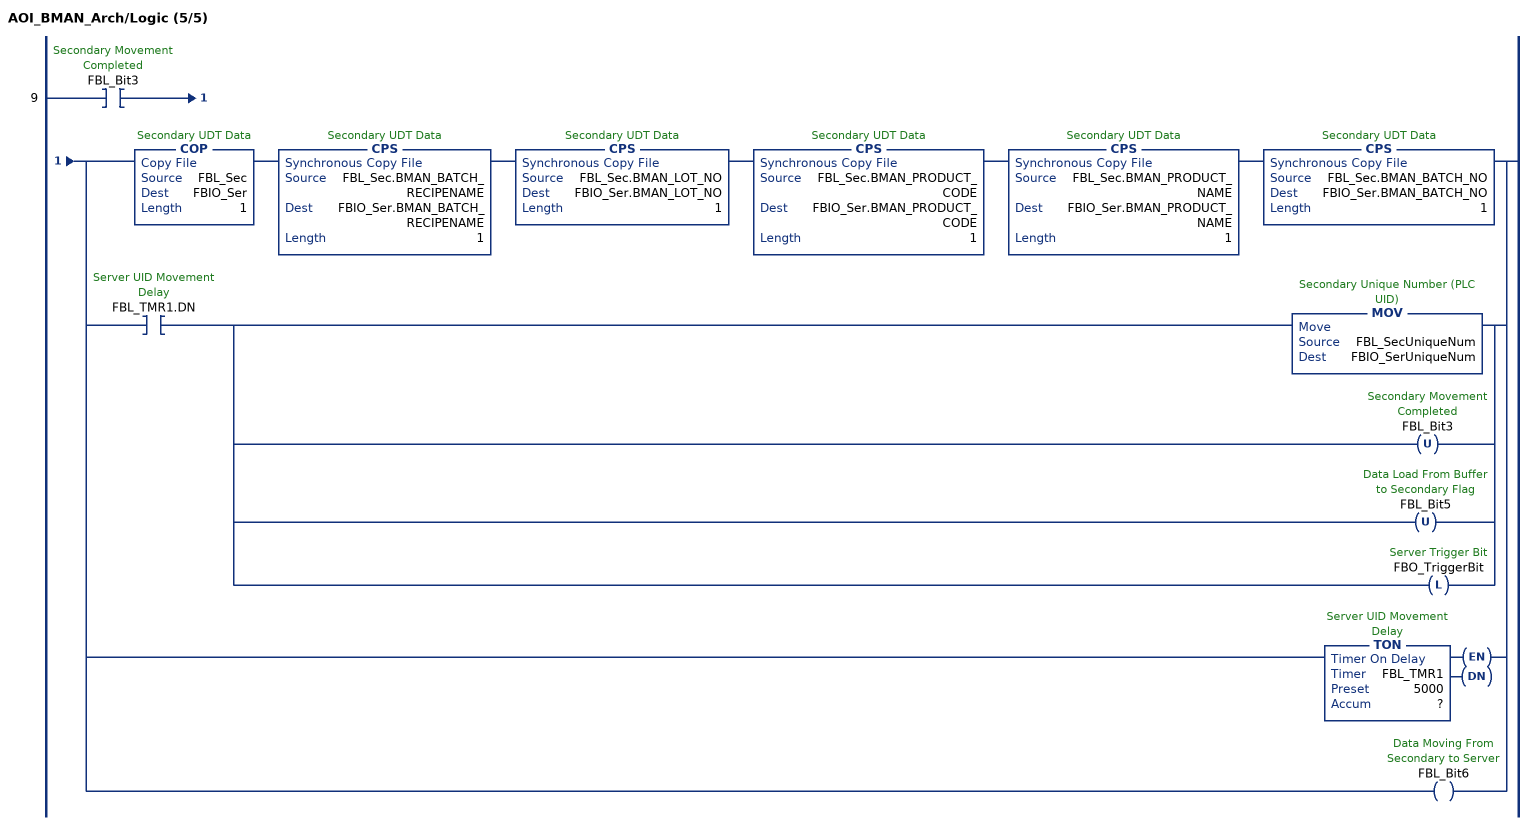
   9: XIC(FBL_Bit3)[COP(FBL_Sec,FBIO_Ser,1) CPS(FBL_Sec.BMAN_BATCH_RECIPENAME,FBIO_Ser.BMAN_BATCH_RECIPENAME,1) CPS(FBL_Sec.BMAN_LOT_NO,FBIO_Ser.BMAN_LOT_NO,1) CPS(FBL_Sec.BMAN_PRODUCT_CODE,FBIO_Ser.BMAN_PRODUCT_CODE,1) CPS(FBL_Sec.BMAN_PRODUCT_NAME,FBIO_Ser.BMAN_PRODUCT_NAME,1) CPS(FBL_Sec.BMAN_BATCH_NO,FBIO_Ser.BMAN_BATCH_NO,1) ,XIC(FBL_TMR1.DN) [MOV(FBL_SecUniqueNum,FBIO_SerUniqueNum) ,OTU(FBL_Bit3) ,OTU(FBL_Bit5) ,OTL(FBO_TriggerBit) ] ,TON(FBL_TMR1,?,?) ,OTE(FBL_Bit6) ];
END_ROUTINE
END_ADD_ON_INSTRUCTION
